PROGRAM Blinker
VAR
	
	fbBlinker1								:FB_Blinker;
	tTurnOffDelayB1							:TIME := T#1S;
	fbBlinker2								:FB_Blinker;
	
END_VAR
(* End *)

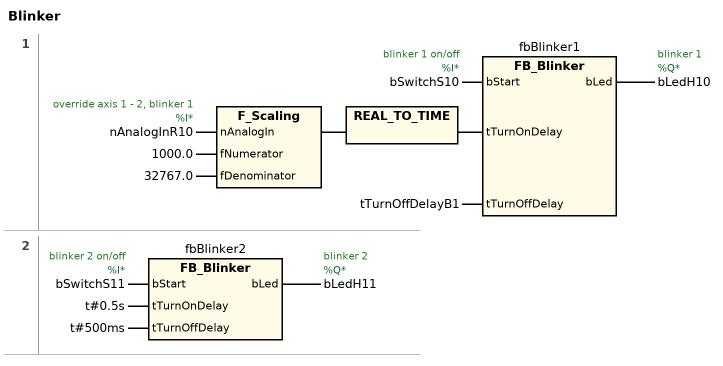
// NETWORK 1
//   bSwitchS10: blinker 1 on/off | AT %I*
//   nAnalogInR10: override axis 1 - 2, blinker 1 | AT %I*
//   bLedH10: blinker 1 | AT %Q*
fbBlinker1(
    bStart := bSwitchS10,
    tTurnOnDelay := REAL_TO_TIME(F_Scaling(nAnalogIn := nAnalogInR10, fNumerator := 1000.0, fDenominator := 32767.0)),
    tTurnOffDelay := tTurnOffDelayB1); // FB_Blinker
bLedH10 := fbBlinker1.bLed;

// NETWORK 2
//   bSwitchS11: blinker 2 on/off | AT %I*
//   bLedH11: blinker 2 | AT %Q*
fbBlinker2(bStart := bSwitchS11, tTurnOnDelay := t#0.5s, tTurnOffDelay := t#500ms); // FB_Blinker
bLedH11 := fbBlinker2.bLed;

END_PROGRAM

(* stored: Version 1.1.0.1, ProductVersion 3.1.4018.5
   POU Blinker: Id {412a77ed-f576-470f-97fb-b89f207e2796}, SpecialFunc None *)
